FUNCTION_BLOCK PAESensorAnalog EXTENDS PAESensorBase
VAR_INPUT
END_VAR
VAR_OUTPUT
END_VAR
VAR
	_ActualValue : LREAL;
	_FaultAckLL1 : BOOL;
	_FaultAckLL2 : BOOL;
	_FaultAckUL1 : BOOL;
	_FaultAckUL2 : BOOL;
	_FaultDelayTimeLL1 : TIME;
	_FaultDelayTimeLL2 : TIME;
	_FaultDelayTimeUL1 : TIME;
	_FaultDelayTimeUL2 : TIME;
	_ForcedSensorValue : LREAL;
	_ForceSensorValue : BOOL;
	_LowerLimit1 : LREAL;
	_LowerLimit2 : LREAL;
	_LowerScaleValue : LREAL;
	_StateLL1 : PANotifyState;
	_StateLL2 : PANotifyState;
	_StateUL1 : PANotifyState;
	_StateUL2 : PANotifyState;
	_UpperLimit1 : LREAL;
	_UpperLimit1Role : PANotifyState;
	_UpperLimit2 : LREAL;
	_UpperLimit2Role : PANotifyState;
	_UpperScaleValue : LREAL;
	_ValueOffset : LREAL;
	_LowerLimit1Role : PAESensorRole;
	_LowerLimit2Role : PAESensorRole;
END_VAR

{attribute 'monitoring' := 'call'}
//{attribute 'TcRpcEnable'}
PROPERTY PUBLIC ActualValue : LREAL
GET // PUBLIC
ActualValue := _ActualValue;
END_GET
SET // PUBLIC
_ActualValue := ActualValue;
Root.OnPropertyChangedLReal(THIS^, 40, _ActualValue);
END_SET
END_PROPERTY

{attribute 'monitoring' := 'call'}
//{attribute 'TcRpcEnable'}
PROPERTY PUBLIC FaultAckLL1 : BOOL
GET // PUBLIC
FaultAckLL1 := _FaultAckLL1;
END_GET
SET // PUBLIC
_FaultAckLL1 := FaultAckLL1;
Root.OnPropertyChangedBool(THIS^, 47, _FaultAckLL1);
END_SET
END_PROPERTY

{attribute 'monitoring' := 'call'}
//{attribute 'TcRpcEnable'}
PROPERTY PUBLIC FaultAckLL2 : BOOL
GET // PUBLIC
FaultAckLL2 := _FaultAckLL2;
END_GET
SET // PUBLIC
_FaultAckLL2 := FaultAckLL2;
Root.OnPropertyChangedBool(THIS^, 48, _FaultAckLL2);
END_SET
END_PROPERTY

{attribute 'monitoring' := 'call'}
//{attribute 'TcRpcEnable'}
PROPERTY PUBLIC FaultAckUL1 : BOOL
GET // PUBLIC
FaultAckUL1 := _FaultAckUL1;
END_GET
SET // PUBLIC
_FaultAckUL1 := FaultAckUL1;
Root.OnPropertyChangedBool(THIS^, 45, _FaultAckUL1);
END_SET
END_PROPERTY

{attribute 'monitoring' := 'call'}
//{attribute 'TcRpcEnable'}
PROPERTY PUBLIC FaultAckUL2 : BOOL
GET // PUBLIC
FaultAckUL2 := _FaultAckUL2;
END_GET
SET // PUBLIC
_FaultAckUL2 := FaultAckUL2;
Root.OnPropertyChangedBool(THIS^, 46, _FaultAckUL2);
END_SET
END_PROPERTY

{attribute 'monitoring' := 'call'}
//{attribute 'TcRpcEnable'}
PROPERTY PUBLIC FaultDelayTimeLL1 : TIME
GET // PUBLIC
FaultDelayTimeLL1 := _FaultDelayTimeLL1;
END_GET
SET // PUBLIC
_FaultDelayTimeLL1 := FaultDelayTimeLL1;
Root.OnPropertyChangedTime(THIS^, 31, _FaultDelayTimeLL1);
END_SET
END_PROPERTY

{attribute 'monitoring' := 'call'}
//{attribute 'TcRpcEnable'}
PROPERTY PUBLIC FaultDelayTimeLL2 : TIME
GET // PUBLIC
FaultDelayTimeLL2 := _FaultDelayTimeLL2;
END_GET
SET // PUBLIC
_FaultDelayTimeLL2 := FaultDelayTimeLL2;
Root.OnPropertyChangedTime(THIS^, 34, _FaultDelayTimeLL2);
END_SET
END_PROPERTY

{attribute 'monitoring' := 'call'}
//{attribute 'TcRpcEnable'}
PROPERTY PUBLIC FaultDelayTimeUL1 : TIME
GET // PUBLIC
FaultDelayTimeUL1 := _FaultDelayTimeUL1;
END_GET
SET // PUBLIC
_FaultDelayTimeUL1 := FaultDelayTimeUL1;
Root.OnPropertyChangedTime(THIS^, 25, _FaultDelayTimeUL1);
END_SET
END_PROPERTY

{attribute 'monitoring' := 'call'}
//{attribute 'TcRpcEnable'}
PROPERTY PUBLIC FaultDelayTimeUL2 : TIME
GET // PUBLIC
FaultDelayTimeUL2 := _FaultDelayTimeUL2;
END_GET
SET // PUBLIC
_FaultDelayTimeUL2 := FaultDelayTimeUL2;	
Root.OnPropertyChangedTime(THIS^, 28, _FaultDelayTimeUL2);
END_SET
END_PROPERTY

METHOD FB_postinit
VAR_INPUT
	root : IACVariobatch;
END_VAR
SUPER^.FB_postinit(root);
root.OnPropertyChangedLReal(THIS^, 23, _UpperLimit1);
root.OnPropertyChangedInt(THIS^, 24, _UpperLimit1Role);
root.OnPropertyChangedTime(THIS^, 25, _FaultDelayTimeUL1);
root.OnPropertyChangedLReal(THIS^, 26, _UpperLimit2);
root.OnPropertyChangedInt(THIS^, 27, _UpperLimit2Role);
root.OnPropertyChangedTime(THIS^, 28, _FaultDelayTimeUL2);
root.OnPropertyChangedLReal(THIS^, 29, _LowerLimit1);
root.OnPropertyChangedInt(THIS^, 30, _LowerLimit1Role);
root.OnPropertyChangedTime(THIS^, 31, _FaultDelayTimeLL1);
root.OnPropertyChangedLReal(THIS^, 32, _LowerLimit2);
root.OnPropertyChangedInt(THIS^, 33, _LowerLimit2Role);
root.OnPropertyChangedTime(THIS^, 34, _FaultDelayTimeLL2);
root.OnPropertyChangedLReal(THIS^, 35, _UpperScaleValue);
root.OnPropertyChangedLReal(THIS^, 36, _LowerScaleValue);
root.OnPropertyChangedLReal(THIS^, 37, _ValueOffset);
root.OnPropertyChangedBool(THIS^, 38, _ForceSensorValue);
root.OnPropertyChangedLReal(THIS^, 39, _ForcedSensorValue);
root.OnPropertyChangedLReal(THIS^, 40, _ActualValue);
root.OnPropertyChangedInt(THIS^, 41, _StateUL1);
root.OnPropertyChangedInt(THIS^, 42, _StateUL2);
root.OnPropertyChangedInt(THIS^, 43, _StateLL1);
root.OnPropertyChangedInt(THIS^, 44, _StateLL2);
root.OnPropertyChangedBool(THIS^, 45, _FaultAckUL1);
root.OnPropertyChangedBool(THIS^, 46, _FaultAckUL2);
root.OnPropertyChangedBool(THIS^, 47, _FaultAckLL1);
root.OnPropertyChangedBool(THIS^, 48, _FaultAckLL2);
END_METHOD

{attribute 'monitoring' := 'call'}
//{attribute 'TcRpcEnable'}
PROPERTY PUBLIC ForcedSensorValue : LREAL
GET // PUBLIC
ForcedSensorValue := _ForcedSensorValue;
END_GET
SET // PUBLIC
_ForcedSensorValue := ForcedSensorValue;
Root.OnPropertyChangedLReal(THIS^, 39, _ForcedSensorValue);
END_SET
END_PROPERTY

{attribute 'monitoring' := 'call'}
//{attribute 'TcRpcEnable'}
PROPERTY PUBLIC ForceSensorValue : BOOL
GET // PUBLIC
ForceSensorValue := _ForceSensorValue;
END_GET
SET // PUBLIC
_ForceSensorValue := ForceSensorValue;
Root.OnPropertyChangedBool(THIS^, 38, _ForceSensorValue);
END_SET
END_PROPERTY

METHOD PUBLIC ForceValue
VAR_INPUT
END_VAR
END_METHOD

METHOD PUBLIC InvokeSetterBool
VAR_INPUT
	PropertyID : INT;
	PropertyValue : BOOL;
END_VAR
SUPER^.InvokeSetterBool(PropertyID, PropertyValue);
CASE PropertyID OF
	38:
		ForceSensorValue := PropertyValue;
	45:
		FaultAckUL1 := PropertyValue;
	46:
		FaultAckUL2 := PropertyValue;
	47:
		FaultAckLL1 := PropertyValue;
	48:
		FaultAckLL2 := PropertyValue;
END_CASE
END_METHOD

METHOD PUBLIC InvokeSetterEnum
VAR_INPUT
	PropertyID : INT;
	PropertyValue : INT;
END_VAR
SUPER^.InvokeSetterEnum(PropertyID, PropertyValue);
CASE PropertyID OF
	30:
		THIS^.LowerLimit1Role := PropertyValue;
	33:
		THIS^.LowerLimit2Role := PropertyValue;
	43:
		THIS^.StateLL1 := PropertyValue;
	44:
		THIS^.StateLL2 := PropertyValue;
	41:
		THIS^.StateUL1 := PropertyValue;
	42:
		THIS^.StateUL2 := PropertyValue;
	24:
		THIS^.UpperLimit1Role := PropertyValue;	
	27:
		THIS^.UpperLimit2Role := PropertyValue;
END_CASE
END_METHOD

METHOD PUBLIC InvokeSetterLReal
VAR_INPUT
	PropertyID : INT;
	PropertyValue : LREAL;
END_VAR
SUPER^.InvokeSetterLReal(PropertyID, PropertyValue);
CASE PropertyID OF
	23:
		UpperLimit1 := PropertyValue;
	26:
		UpperLimit2 := PropertyValue;
	29:
		LowerLimit1 := PropertyValue;
	32:
		LowerLimit2 := PropertyValue;
	35:
		UpperScaleValue := PropertyValue;
	36:
		LowerScaleValue := PropertyValue;
	37:
		ValueOffset := PropertyValue;
	39:
		ForcedSensorValue := PropertyValue;
	40:
		ActualValue := PropertyValue;
END_CASE
END_METHOD

METHOD PUBLIC InvokeSetterTime
VAR_INPUT
	PropertyID : INT;
	PropertyValue : DINT;
END_VAR
SUPER^.InvokeSetterTime(PropertyID, PropertyValue);
CASE PropertyID OF
	25:
		FaultDelayTimeUL1 := TO_TIME(PropertyValue);
	28:
		FaultDelayTimeUL2 := TO_TIME(PropertyValue);
	31:
		FaultDelayTimeLL1 := TO_TIME(PropertyValue);
	34:
		FaultDelayTimeLL2 := TO_TIME(PropertyValue);	
END_CASE
END_METHOD

METHOD PUBLIC IsEnabledAcknowledgeAlarms : BOOL
VAR_INPUT
END_VAR
END_METHOD

METHOD PUBLIC IsEnabledForceValue : BOOL
VAR_INPUT
END_VAR
END_METHOD

METHOD PUBLIC IsEnabledResetValue : BOOL
VAR_INPUT
END_VAR
END_METHOD

{attribute 'monitoring' := 'call'}
//{attribute 'TcRpcEnable'}
PROPERTY PUBLIC LowerLimit1 : LREAL
GET // PUBLIC
LowerLimit1:=_LowerLimit1;
END_GET
SET // PUBLIC
_LowerLimit1 := LowerLimit1;
Root.OnPropertyChangedLReal(THIS^, 29, _LowerLimit1);
END_SET
END_PROPERTY

{attribute 'monitoring' := 'call'}
//{attribute 'TcRpcEnable'}
PROPERTY PUBLIC LowerLimit1Role : PAESensorRole
GET // PUBLIC
LowerLimit1Role := _LowerLimit1Role;
END_GET
SET // PUBLIC
_LowerLimit1Role := LowerLimit1Role;
Root.OnPropertyChangedInt(THIS^, 30, _LowerLimit1Role);
END_SET
END_PROPERTY

{attribute 'monitoring' := 'call'}
//{attribute 'TcRpcEnable'}
PROPERTY PUBLIC LowerLimit2 : LREAL
GET // PUBLIC
LowerLimit2 := _LowerLimit2;
END_GET
SET // PUBLIC
_LowerLimit2 := LowerLimit2;
Root.OnPropertyChangedLReal(THIS^, 32, _LowerLimit2);
END_SET
END_PROPERTY

{attribute 'monitoring' := 'call'}
//{attribute 'TcRpcEnable'}
PROPERTY PUBLIC LowerLimit2Role : PAESensorRole
GET // PUBLIC
LowerLimit2Role := _LowerLimit2Role;
END_GET
SET // PUBLIC
_LowerLimit2Role := LowerLimit2Role;
Root.OnPropertyChangedInt(THIS^, 33, _LowerLimit2Role);
END_SET
END_PROPERTY

{attribute 'monitoring' := 'call'}
//{attribute 'TcRpcEnable'}
PROPERTY PUBLIC LowerScaleValue : LREAL
GET // PUBLIC
LowerScaleValue := _LowerScaleValue;
END_GET
SET // PUBLIC
_LowerScaleValue := LowerScaleValue;
Root.OnPropertyChangedLReal(THIS^, 36, _LowerScaleValue);
END_SET
END_PROPERTY

METHOD OnInitMemory
VAR_INPUT
	root : IACVariobatch;
END_VAR
RegisterProperty(root, 23, GCL.cSizeLREAL); //UpperLimit1
RegisterProperty(root, 24, GCL.cSizeINT); //UpperLimit1Role
RegisterProperty(root, 25, GCL.cSizeTIME); //FaultDelayTimeUL1
RegisterProperty(root, 26, GCL.cSizeLREAL); //UpperLimit2
RegisterProperty(root, 27, GCL.cSizeINT); //UpperLimit2Role
RegisterProperty(root, 28, GCL.cSizeTIME); //FaultDelayTimeUL2
RegisterProperty(root, 29, GCL.cSizeLREAL); //LowerLimit1
RegisterProperty(root, 30, GCL.cSizeINT); //LowerLimit1Role
RegisterProperty(root, 31, GCL.cSizeTIME); //FaultDelayTimeLL1
RegisterProperty(root, 32, GCL.cSizeLREAL); //LowerLimit2
RegisterProperty(root, 33, GCL.cSizeINT); //LowerLimit2Role
RegisterProperty(root, 34, GCL.cSizeTIME); //FaultDelayTimeLL2
RegisterProperty(root, 35, GCL.cSizeLREAL); //UpperScaleValue
RegisterProperty(root, 36, GCL.cSizeLREAL); //LowerScaleValue
RegisterProperty(root, 37, GCL.cSizeLREAL); //ValueOffset
RegisterProperty(root, 38, GCL.cSizeBYTE); //ForceSensorvalue
RegisterProperty(root, 39, GCL.cSizeLREAL); //ForcedSensorValue
RegisterProperty(root, 40, GCL.cSizeLREAL); //ActualValue
RegisterProperty(root, 41, GCL.cSizeINT); //StateUL1
RegisterProperty(root, 42, GCL.cSizeINT); //StateUL2
RegisterProperty(root, 43, GCL.cSizeINT); //StateLL1
RegisterProperty(root, 44, GCL.cSizeINT); //StateLL2
RegisterProperty(root, 45, GCL.cSizeBYTE); //FaultAckUL1
RegisterProperty(root, 46, GCL.cSizeBYTE); //FaultAckUL2
RegisterProperty(root, 47, GCL.cSizeBYTE); //FaultAckLL1
RegisterProperty(root, 48, GCL.cSizeBYTE); //FaultAckLL2
SUPER^.OnInitMemory(root);
END_METHOD

METHOD PUBLIC OnSetStateLL1
VAR_INPUT
END_VAR
END_METHOD

METHOD PUBLIC OnSetStateLL2
VAR_INPUT
END_VAR
END_METHOD

METHOD PUBLIC OnSetStateUL1
VAR_INPUT
END_VAR
END_METHOD

METHOD PUBLIC OnSetStateUL2
VAR_INPUT
END_VAR
END_METHOD

METHOD PUBLIC PAESensorAnalog
VAR_INPUT
END_VAR
END_METHOD

METHOD PUBLIC ResetValue
VAR_INPUT
END_VAR
END_METHOD

{attribute 'monitoring' := 'call'}
//{attribute 'TcRpcEnable'}
PROPERTY PUBLIC StateLL1 : PANotifyState
GET // PUBLIC
StateLL1 := _StateLL1;
END_GET
SET // PUBLIC
_StateLL1 := StateLL1;
Root.OnPropertyChangedInt(THIS^, 43, _StateLL1);
END_SET
END_PROPERTY

METHOD StateLL1_PropertyChanged
VAR_INPUT
END_VAR
END_METHOD

{attribute 'monitoring' := 'call'}
//{attribute 'TcRpcEnable'}
PROPERTY PUBLIC StateLL2 : PANotifyState
GET // PUBLIC
StateLL2 := _StateLL2;
END_GET
SET // PUBLIC
_StateLL2 := StateLL2;
Root.OnPropertyChangedInt(THIS^, 44, _StateLL2);
END_SET
END_PROPERTY

METHOD StateLL2_PropertyChanged
VAR_INPUT
END_VAR
END_METHOD

{attribute 'monitoring' := 'call'}
//{attribute 'TcRpcEnable'}
PROPERTY PUBLIC StateUL1 : PANotifyState
GET // PUBLIC
StateUL1 := _StateUL1;
END_GET
SET // PUBLIC
_StateUL1 := StateUL1;
Root.OnPropertyChangedInt(THIS^, 41, _StateUL1);
END_SET
END_PROPERTY

METHOD StateUL1_PropertyChanged
VAR_INPUT
END_VAR
END_METHOD

{attribute 'monitoring' := 'call'}
//{attribute 'TcRpcEnable'}
PROPERTY PUBLIC StateUL2 : PANotifyState
GET // PUBLIC
StateUL2 := _StateUL2;
END_GET
SET // PUBLIC
_StateUL2 := StateUL2;
Root.OnPropertyChangedInt(THIS^, 42, _StateUL2);
END_SET
END_PROPERTY

METHOD StateUL2_PropertyChanged
VAR_INPUT
END_VAR
END_METHOD

{attribute 'monitoring' := 'call'}
//{attribute 'TcRpcEnable'}
PROPERTY PUBLIC UpperLimit1 : LREAL
GET // PUBLIC
UpperLimit1 := _UpperLimit1;
END_GET
SET // PUBLIC
_UpperLimit1 := UpperLimit1;
Root.OnPropertyChangedLReal(THIS^, 23, _UpperLimit1);
END_SET
END_PROPERTY

{attribute 'monitoring' := 'call'}
//{attribute 'TcRpcEnable'}
PROPERTY PUBLIC UpperLimit1Role : PANotifyState
GET // PUBLIC
UpperLimit1Role := _UpperLimit1Role;
END_GET
SET // PUBLIC
_UpperLimit1Role := UpperLimit1Role;
Root.OnPropertyChangedInt(THIS^, 24, _UpperLimit1Role);
END_SET
END_PROPERTY

{attribute 'monitoring' := 'call'}
//{attribute 'TcRpcEnable'}
PROPERTY PUBLIC UpperLimit2 : LREAL
GET // PUBLIC
UpperLimit2 := _UpperLimit2;
END_GET
SET // PUBLIC
_UpperLimit2 := UpperLimit2;
Root.OnPropertyChangedLReal(THIS^, 26, _UpperLimit2);
END_SET
END_PROPERTY

{attribute 'monitoring' := 'call'}
//{attribute 'TcRpcEnable'}
PROPERTY PUBLIC UpperLimit2Role : PANotifyState
GET // PUBLIC
UpperLimit2Role := _UpperLimit2Role;
END_GET
SET // PUBLIC
_UpperLimit2Role := UpperLimit2Role;
Root.OnPropertyChangedInt(THIS^, 27, _UpperLimit2Role);
END_SET
END_PROPERTY

{attribute 'monitoring' := 'call'}
//{attribute 'TcRpcEnable'}
PROPERTY PUBLIC UpperScaleValue : LREAL
GET // PUBLIC
UpperScaleValue := _UpperScaleValue;
END_GET
SET // PUBLIC
_UpperScaleValue := UpperScaleValue;
Root.OnPropertyChangedLReal(THIS^, 35, _UpperScaleValue);
END_SET
END_PROPERTY

{attribute 'monitoring' := 'call'}
//{attribute 'TcRpcEnable'}
PROPERTY PUBLIC ValueOffset : LREAL
GET // PUBLIC
ValueOffset := _ValueOffset;
END_GET
SET // PUBLIC
_ValueOffset := ValueOffset;
Root.OnPropertyChangedLReal(THIS^, 37, _ValueOffset);
END_SET
END_PROPERTY

END_FUNCTION_BLOCK

(* stored: Version 1.1.0.1, ProductVersion 3.1.4024.6
   POU PAESensorAnalog: Id {94b8ea30-db6c-4d72-920b-3b65a6203388}, SpecialFunc None
   Property ActualValue: Id {0caf50f3-e2fa-4463-8b05-e1ab93f3cf6d}
   Get Get: Id {32394500-ff71-47a7-b9aa-cf8b3444caa6}
   Set Set: Id {0d6ba7b1-c6de-44ea-b65d-14de2f7819a7}
   Property FaultAckLL1: Id {37ac2df0-e3b3-4e93-ba0e-2f9bc976e345}
   Get Get: Id {2da072a4-d361-487c-9518-54d68c13be8e}
   Set Set: Id {8547b351-195e-4c92-b3a1-b96c4ff7c7e2}
   Property FaultAckLL2: Id {5e7e8f9c-3a42-4d06-90f2-13919a3b2098}
   Get Get: Id {e374b049-874f-4cc4-b6e7-eddf5ff54a0d}
   Set Set: Id {98107545-aa14-4b29-b981-d5de29d61ca6}
   Property FaultAckUL1: Id {31ed7923-1b79-4b3e-b5d3-0788d282e274}
   Get Get: Id {a33cb09c-eb99-4823-88df-ab511cf97a43}
   Set Set: Id {ff9399de-46ce-4092-8134-d27bd7cf3656}
   Property FaultAckUL2: Id {d6ae1e1e-de20-4dc7-9c8c-2018a576c7ae}
   Get Get: Id {6ed1c7b0-eed4-4067-8826-8d67f681bccd}
   Set Set: Id {ee5afb6c-d2ad-47b5-8578-27b8e7afc56c}
   Property FaultDelayTimeLL1: Id {d46771c0-ab3b-4f0c-9c6f-55f93864196f}
   Get Get: Id {18f3e3a5-c97d-4a93-bc4a-61fef93ca5bd}
   Set Set: Id {832c09b8-99a4-4360-be06-5196b52a9f16}
   Property FaultDelayTimeLL2: Id {5a9cab5c-6a8a-4862-a936-a3be2f74efba}
   Get Get: Id {721180a9-f89e-4537-bbf9-06b95631c34c}
   Set Set: Id {408dd4b3-81ea-4f85-a9e6-ddfa4daec4b5}
   Property FaultDelayTimeUL1: Id {a5bba629-110c-4dc7-a2c9-80f306e657c7}
   Get Get: Id {fb832f11-6fc4-4255-87dc-f1ffe006dc84}
   Set Set: Id {2060c70f-4cdb-4c08-83b0-29f7ed11170e}
   Property FaultDelayTimeUL2: Id {1efbe7dd-2672-4818-8a85-76ee7b1cc3d5}
   Get Get: Id {d2575855-dfe1-4257-8f36-a16ba57ccf53}
   Set Set: Id {153f5850-85be-49a1-ae87-0f6f0ade1a39}
   Method FB_postinit: Id {e204d4af-cbbc-482f-8bcc-63a07d84218e}
   Property ForcedSensorValue: Id {43289bd4-9be2-4d98-b0fd-d1421fd0e3ef}
   Get Get: Id {29c5ebc8-82f4-44e9-82b2-35e0d34c77b9}
   Set Set: Id {78bd5c38-f5bf-49b4-b0e0-819493a75880}
   Property ForceSensorValue: Id {85f68740-b81e-4970-a07c-318fd114d695}
   Get Get: Id {2e6455ff-cb9a-49a3-9063-3ae9d235ab70}
   Set Set: Id {bb2acca3-6eb4-42c6-be10-9e4bfaa9ee2d}
   Method ForceValue: Id {07bdbaa0-c794-4716-8d9a-3cf4ee43f92f}
   Method InvokeSetterBool: Id {1db5267f-c17c-492d-889c-e204803c0f4b}
   Method InvokeSetterEnum: Id {b6963973-157a-40ca-98fa-37c7f0dcfcea}
   Method InvokeSetterLReal: Id {c47f0698-9baf-454f-b674-f1690743cdac}
   Method InvokeSetterTime: Id {17188ee8-923d-47a9-b7de-304d37441be0}
   Method IsEnabledAcknowledgeAlarms: Id {6712f1d9-5e31-45a1-9f2e-12bb65237f93}
   Method IsEnabledForceValue: Id {1ecef7ba-fc54-4fd8-beb5-0037d810d853}
   Method IsEnabledResetValue: Id {46cc8f7e-f427-4657-868f-4683cd78c666}
   Property LowerLimit1: Id {604c12c0-45d7-433d-85ef-4ad80545d590}
   Get Get: Id {fcfb3723-7a09-4c0a-a711-c1692a94536b}
   Set Set: Id {f7499f1b-1e7b-49b5-98d8-0defde4ad95c}
   Property LowerLimit1Role: Id {1dc216a6-54c1-4fa0-85fd-d50c2f304a3d}
   Get Get: Id {6abae84b-b3c5-457b-b850-f7e89019292e}
   Set Set: Id {dba687d9-9462-4e34-adbc-d642719b7696}
   Property LowerLimit2: Id {f965f486-4d23-418a-be89-155824e88d13}
   Get Get: Id {8e5cead0-3c20-4969-a120-2fbf5bb3a01a}
   Set Set: Id {7bc7a352-b653-4514-a3f7-e4d9f730d6a1}
   Property LowerLimit2Role: Id {fd53466d-74ff-4579-b1e3-1d2b2c80e58f}
   Get Get: Id {4ccfce3e-10aa-48f5-9123-58b7fd34f5a3}
   Set Set: Id {0609f35d-9cb0-4017-bd01-e9e81ae5b78c}
   Property LowerScaleValue: Id {6e049d43-3d0b-495f-91a5-371a55a236dd}
   Get Get: Id {d265cb53-e71d-4449-9a99-2ae482e8fbe8}
   Set Set: Id {b5943a91-3789-4913-99ee-f176d0078bfd}
   Method OnInitMemory: Id {44f578e5-ae8e-42d4-b89b-30ccbd3325c5}
   Method OnSetStateLL1: Id {6e88bceb-368f-4daf-a814-dbd1481f1e78}
   Method OnSetStateLL2: Id {6fe795ce-b074-4e80-87aa-dd7224de9d8c}
   Method OnSetStateUL1: Id {9ed249f3-945b-4748-bff2-6d225bc638d6}
   Method OnSetStateUL2: Id {0a804a32-7358-40c2-a36d-3d2dfc26d8ef}
   Method PAESensorAnalog: Id {270ba104-13b4-41b3-ac95-ea419776e93d}
   Method ResetValue: Id {255da4a5-8311-4068-ada0-8f6b99bace08}
   Property StateLL1: Id {43fc4e96-4d6c-40d6-93df-4638e49f3e2d}
   Get Get: Id {eb2e4d1a-d0af-41ce-a560-ab19c8cd3084}
   Set Set: Id {c9f52310-4970-499e-9574-a23947c9c087}
   Method StateLL1_PropertyChanged: Id {5a004be5-de93-4ded-9ccb-6261ee09f5df}
   Property StateLL2: Id {bde90643-1e63-4425-bfb8-407c31f2dfc5}
   Get Get: Id {96592b01-e159-472e-995c-0315ce60da7b}
   Set Set: Id {2f087758-4c14-4a37-b71b-0fce3b1b0cb0}
   Method StateLL2_PropertyChanged: Id {bb08b218-8539-40de-9f20-42596efe7a0e}
   Property StateUL1: Id {371c491a-26c0-4ae9-b3b9-9d7dae4372d4}
   Get Get: Id {bb38e161-00d8-4e72-bc88-92320adf35e4}
   Set Set: Id {3be0be1a-b436-4fcf-9c53-fd12a12edd6b}
   Method StateUL1_PropertyChanged: Id {b281e056-5d6a-4ec8-baae-9afb209a8529}
   Property StateUL2: Id {ba167bdb-6306-4e0f-8ccd-4b615643acf6}
   Get Get: Id {7a2b71a5-f561-466b-9597-d6ea0ce4415a}
   Set Set: Id {6615c7fc-74c2-475d-9eef-a1f6ed85cb4b}
   Method StateUL2_PropertyChanged: Id {8b66b88c-53fd-4d1b-82f0-e3a9d1c5b8b5}
   Property UpperLimit1: Id {c2a87e39-3fdd-4c21-b4d5-b3ee70a0b9cf}
   Get Get: Id {6ee94690-f536-48a5-b7b1-0f15aa914b2c}
   Set Set: Id {d1a61991-60a8-4340-987b-37279afb6897}
   Property UpperLimit1Role: Id {ea4ffaa1-033b-4f15-9272-35493cb77e8b}
   Get Get: Id {739285e6-282b-499a-ab25-ba9b08528f6a}
   Set Set: Id {43cdcce5-b3f6-4056-bec9-de009560d307}
   Property UpperLimit2: Id {f9b5d045-acc2-43bc-9747-36cca3ce78cc}
   Get Get: Id {f26b0ea8-6dae-48ba-b82a-a543d84b8c41}
   Set Set: Id {3216360b-4627-47ee-b5c0-bc035f14f1dc}
   Property UpperLimit2Role: Id {1dc75716-529a-40cf-b30e-27b4e79c23a5}
   Get Get: Id {0ff78972-eee7-444e-8033-1f31fcc1cdc5}
   Set Set: Id {ca37f434-766f-4f95-8804-4d5569ab15c1}
   Property UpperScaleValue: Id {07e630f8-8263-452f-b944-9a6e8a9b4f72}
   Get Get: Id {c4be7d71-b1d4-4bff-88ea-c1f5b8636c73}
   Set Set: Id {5d6f852c-7d43-477d-850e-0b3b1b7b4ce0}
   Property ValueOffset: Id {752a1df6-bbae-4a95-8158-af8f56765fef}
   Get Get: Id {ea90bd66-8250-4082-8b9c-09558bc9ceaa}
   Set Set: Id {c88f1de6-af65-4501-892b-748af4cb4380} *)
